Fanuc KAREL source: kd00030.KL

-- PROVISIONAL review KL for V1013-1; original PC SHA256 4b29c8843c7b2464827457ee780287ac422c2a7e70e1000c17b0c72f82b794e6
-- Incomplete behavior may be omitted. Consult companion uncertainty JSON. Do not deploy.
PROGRAM KD00030
%NOLOCKGROUP
VAR
  I : INTEGER
  J : INTEGER
  B : BOOLEAN
  R : REAL
  S : STRING[80]
BEGIN
  -- UNRESOLVED_PC offsets 5-21; opcodes 9D,81,18,9C,12,22,9D,13,04
  -- UNRESOLVED_PC offsets 26-30; opcodes 7F
END KD00030
